RoboDK station: practica1i2TercerIntento.rdk

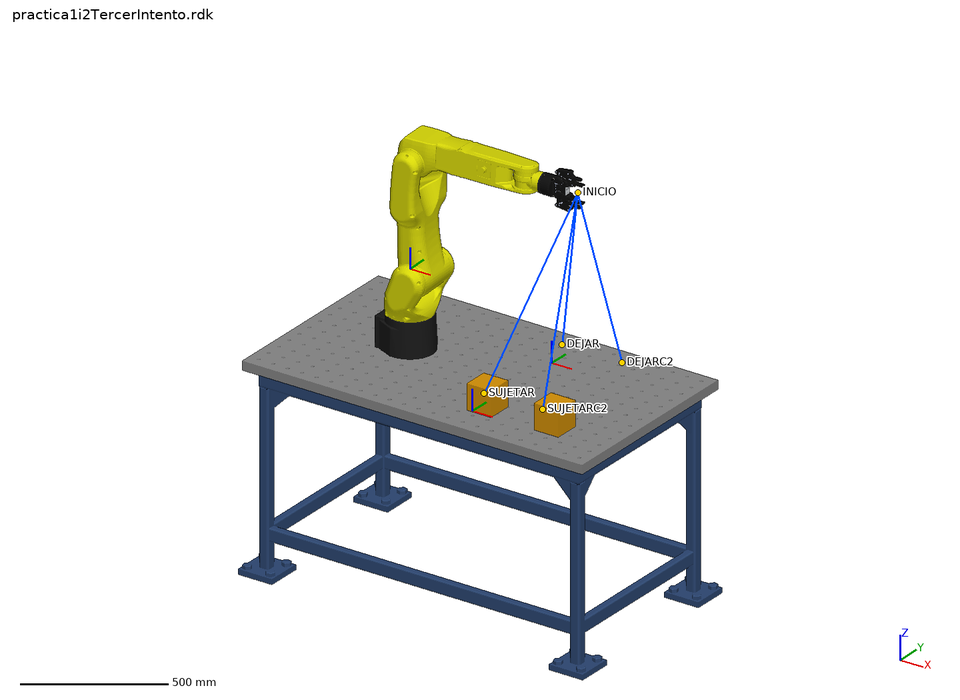
[picture v0: the station drawn from its stored meshes, robots at their saved joint values, targets as dots, program paths as lines]
Station practica1i2TercerIntento (saved by RoboDK 6.0.0). Poses are relative to the parent item; angles as X-Y-Z fixed-axis rotations.
  - object Table 1400x800x800mm at (0, 0, 0) mm, size 1420 x 820 x 800 mm, geometry from Table-1400x800x800mm.sld
  - frame Fanuc LR Mate 200iD/7L Base at (70.2, 3.67, 297.49) mm, rotated rx 0.7 ry 0.59 rz 1.98 deg
    - robot Fanuc LR Mate 200iD/7L: 6 axes, payload 7 kg, reach 911 mm, repeatability 0.01 mm, weight 27 kg
        modified DH rows (alpha deg, a mm, theta deg, d mm): 0, 0, 0, 330; -90, 50, -90, 0; 0, 440, 0, 0; -90, 35, 0, 420; 90, 0, 0, 0; -90, 0, 0, 80
        base shift (0, 0, -330) mm
        joint limits [-180, -100, -150, -190, -125, -360] to [180, 145, 280, 190, 125, 360]; home [0, 0, 0, 0, 0, 0]; saved at [0.03, -0.915, -0.003, -85.166, 0, 85.167]
      - tool RobotiQ 2F-85 Gripper (Open), TCP at (0, 0, 130) mm, size 147.4 x 75 x 146.8 mm
      - tool RobotiQ 2F-85 Gripper (Closed), TCP at (0, 0, 130) mm, size 134.4 x 75 x 157.6 mm
  - frame PICK at (538.36, -298.62, 16) mm
    - object 2do cubo at (256.59, -5.91, 4.25) mm, size 100 x 100 x 100 mm, geometry from Cube-100mm.sld
    - target INICIO (Cartesian target) at (209.42, 320.17, 749.47) mm, rotated rx -129.84 ry -89.09 rz -48.18 deg; joints [0, 0, 0, 0, 0, 0] of Fanuc LR Mate 200iD/7L
    - target SUJETAR (Cartesian target) at (12.7, 50.77, 49.71) mm, rotated rx -129.84 ry -89.09 rz -48.19 deg; joints [-45.702, 64.071, -103.964, 46.561, 99.703, 10.092] of Fanuc LR Mate 200iD/7L
    - target DEJAR (Cartesian target) at (20.99, 496.7, 56.53) mm, rotated rx -129.83 ry -89.09 rz -48.19 deg; joints [31.247, 65.282, -110.313, -32.902, 107.265, -10.87] of Fanuc LR Mate 200iD/7L
    - target SUJETARC2 (Cartesian target) at (255.2, 49.8, 57.09) mm, rotated rx -129.84 ry -89.09 rz -48.18 deg; joints [-28.938, 64.836, -76.731, 29.599, 78.413, -6.509] of Fanuc LR Mate 200iD/7L
    - target DEJARC2 (Cartesian target) at (269.77, 494.57, 58.67) mm, rotated rx -129.84 ry -89.09 rz -48.18 deg; joints [16.998, 64.606, -79.154, -17.289, 79.634, 3.206] of Fanuc LR Mate 200iD/7L
    - object 1er cubo at (5.29, -42.51, 22.82) mm, size 100 x 100 x 100 mm, geometry from Cube-100mm.sld
  - frame PLACE at (547.88, 151.77, 19.41) mm
  - program Prog1 (15 instructions, listed below)
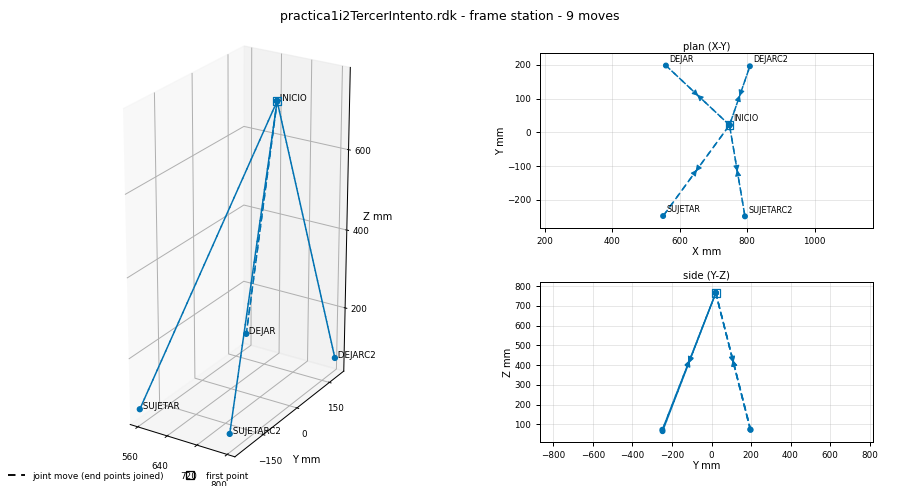
[picture p0: tool path of practica1i2TercerIntento.rdk in frame station, 9 of 9 moves have a stored position in this frame; points joined in program order, loops and branches not executed]

--- program Prog1 (robot Fanuc LR Mate 200iD/7L) ---
  Est. Ref.: PICK
  Est. herr: RobotiQ 2F-85 Gripper (Open)
  MoveJ (INICIO)
  MoveJ (SUJETAR)
  Adjuntar a RobotiQ 2F-85 Gripper (Open)
  MoveJ (INICIO)
  MoveJ (DEJAR)
  Separar de RobotiQ 2F-85 Gripper (Open)
  MoveJ (INICIO)
  MoveJ (SUJETARC2)
  Adjuntar a RobotiQ 2F-85 Gripper (Open)
  MoveJ (INICIO)
  MoveJ (DEJARC2)
  Separar de RobotiQ 2F-85 Gripper (Open)
  MoveJ (INICIO)
